(* IEC 61131-3 sources: STruCpp/tests/st-validation/data_types, 28 files *)

(* ---- string_conversions.st ---- *)
FUNCTION_BLOCK StringConversions
  VAR_OUTPUT
    (* STRING numeric parsers — strtol / strtoul / strtod under the hood,
       so `'3.14'` parses to 3 as an integer (strtol stops at the '.')
       and to 3.14 as a REAL. *)
    str_to_uint    : UINT;
    str_to_int     : INT;
    str_to_dint    : DINT;
    str_to_lint    : LINT;
    str_to_real    : REAL;
    str_to_lreal   : LREAL;
    str_negative   : INT;
    str_hex_skip   : UINT;
    str_bool_true  : BOOL;
    str_bool_false : BOOL;

    (* WSTRING numeric parsers — route through WSTRING_TO_STRING so the
       parse rules stay byte-identical with the STRING path.  Anything
       beyond the ASCII numeric subset is the user's responsibility
       (the transcoder truncates to the low byte). *)
    wstr_to_uint : UINT;
    wstr_to_real : LREAL;
    wstr_to_bool : BOOL;
  END_VAR
  VAR
    s_pi      : STRING := '3.14';
    s_half    : STRING := '4.5';
    s_neg     : STRING := '-42';
    s_trail   : STRING := '12abc';
    s_true    : STRING := 'TRUE';
    s_false   : STRING := 'no';
    ws_pi     : WSTRING := "3.14";
    ws_true   : WSTRING := "true";
  END_VAR

  str_to_uint    := TO_UINT(s_pi);     (* 3   — strtoul stops at '.' *)
  str_to_int     := TO_INT(s_pi);      (* 3 *)
  str_to_dint    := TO_DINT(s_pi);     (* 3 *)
  str_to_lint    := TO_LINT(s_pi);     (* 3 *)
  (* `3.14` round-trips bit-exact through LREAL (double) but loses
     precision narrowing to REAL (float).  Test framework's ASSERT_EQ
     does bit-exact float compare, so use an exactly-representable
     fraction here (`4.5` = 9/2 = exact in IEEE-754) instead of `3.14`. *)
  str_to_real    := TO_REAL(s_half);   (* 4.5 *)
  str_to_lreal   := TO_LREAL(s_pi);    (* 3.14 *)
  str_negative   := TO_INT(s_neg);     (* -42 *)
  str_hex_skip   := TO_UINT(s_trail);  (* 12  — strtoul stops at 'a' *)
  str_bool_true  := TO_BOOL(s_true);   (* TRUE *)
  str_bool_false := TO_BOOL(s_false);  (* FALSE *)

  wstr_to_uint := TO_UINT(ws_pi);    (* 3 *)
  wstr_to_real := TO_LREAL(ws_pi);   (* 3.14 *)
  wstr_to_bool := TO_BOOL(ws_true);  (* TRUE *)
END_FUNCTION_BLOCK

(* ---- strings.st ---- *)
FUNCTION_BLOCK StringHolder
  VAR_OUTPUT
    dblQuote : STRING;
    apostrophe : STRING;
    backslash : STRING;
    dblQuoteLen : INT;
    apostropheLen : INT;
    backslashLen : INT;
  END_VAR
  dblQuote := 'say "hello"';
  apostrophe := 'it''s working';
  backslash := 'C:\\Users\\test';
  dblQuoteLen := LEN(dblQuote);
  apostropheLen := LEN(apostrophe);
  backslashLen := LEN(backslash);
END_FUNCTION_BLOCK

(* ---- time_types.st ---- *)
FUNCTION_BLOCK TimeConversions
  VAR_OUTPUT
    (* TIME → integer scales ns→ms *)
    ms_via_dint  : DINT;
    ms_via_uint  : UINT;
    ms_via_real  : REAL;

    (* Explicit TIME_TO_<unit> helpers still work and pick the unit
       the user names, regardless of the generic TO_<int>(TIME) ms
       default.  TIME_TO_US returns LINT (int64_t) on the runtime
       side — declared wide enough to receive the raw value without
       a narrowing assignment.  Names are prefixed `unit_` so they
       don't shadow the runtime helper names on the RHS. *)
    unit_us      : LINT;
    unit_seconds : LREAL;

    (* TOD → integer scales ns→ms (since midnight) *)
    tod_ms       : DINT;

    (* DT → integer is SECONDS since 1970-01-01, matching CODESYS:
       DT_TO_DINT(DT#2019-9-1-12:0:0.0) = 1567339200.  Kept in LINT so the
       assertion reads the value rather than a truncation of it. *)
    dt_seconds   : LINT;

    (* DATE → integer is SECONDS too — CODESYS keeps DATE in DT's memory
       format, so DATE_TO_DINT(D#1970-1-2) = 86400, not 1.  UDINT rather
       than UINT: a day count fits 16 bits, a second count does not, and
       the old UINT declaration was quietly asserting a 16-bit truncation. *)
    date_seconds : UDINT;
  END_VAR
  VAR
    duration : TIME := T#1500ms;
    midpoint : TOD  := TOD#06:00:00;
    moment   : DT   := DT#1970-01-01-00:00:01;
    day      : DATE := DATE#1970-01-15;
  END_VAR

  ms_via_dint  := TIME_TO_DINT(duration);   (* 1500 *)
  ms_via_uint  := TIME_TO_UINT(duration);   (* 1500 *)
  ms_via_real  := TIME_TO_REAL(duration);   (* 1500.0 *)
  unit_us      := TIME_TO_US(duration);     (* 1_500_000 *)
  unit_seconds := TIME_TO_S(duration);      (* 1.5 *)

  tod_ms    := TOD_TO_DINT(midpoint);   (* 21_600_000 — 6h in ms *)
  dt_seconds   := TO_LINT(moment);      (* 1 — one second after the epoch *)
  date_seconds := TO_UDINT(day);        (* 1209600 — 14 days, in seconds *)
END_FUNCTION_BLOCK

(* ---- arrays.st ---- *)
TYPE IntArray : ARRAY[1..5] OF INT; END_TYPE

PROGRAM ArrayTest
  VAR
    arr : IntArray;
    sum : INT;
    first : INT;
    last : INT;
    i : INT;
  END_VAR

  (* Initialize array *)
  FOR i := 1 TO 5 DO
    arr[i] := i * 10;
  END_FOR;

  first := arr[1];
  last := arr[5];

  (* Sum all elements *)
  sum := 0;
  FOR i := 1 TO 5 DO
    sum := sum + arr[i];
  END_FOR;
END_PROGRAM

(* ---- booleans.st ---- *)
PROGRAM BooleanTypeTest
  VAR
    t : BOOL;
    f : BOOL;
    and_tt : BOOL;
    and_tf : BOOL;
    or_ff : BOOL;
    or_tf : BOOL;
    not_t : BOOL;
    not_f : BOOL;
  END_VAR

  t := TRUE;
  f := FALSE;
  and_tt := t AND t;
  and_tf := t AND f;
  or_ff := f OR f;
  or_tf := t OR f;
  not_t := NOT t;
  not_f := NOT f;
END_PROGRAM

(* ---- enum_bare_members.st ---- *)
TYPE
  TrafficState : (RED, YELLOW, GREEN);
  PedestrianState : (WALK, DONT_WALK, FLASHING);
END_TYPE

PROGRAM EnumBareTest
  VAR_INPUT
    ts : TrafficState := RED;
    ps : PedestrianState := WALK;
  END_VAR
  VAR
    result   : INT;
    isRed    : BOOL;
    isWalk   : BOOL;
  END_VAR

  (* Bare enum comparison *)
  isRed := (ts = RED);
  isWalk := (ps = WALK);

  (* CASE with bare enum labels *)
  CASE ts OF
    RED:
      result := 1;
    GREEN:
      result := 2;
    YELLOW:
      result := 3;
  END_CASE;
END_PROGRAM

(* ---- enum_dot_notation.st ---- *)
TYPE
  TrafficState : (RED, YELLOW, GREEN);
  PedestrianState : (WALK, DONT_WALK, FLASHING);
END_TYPE

PROGRAM EnumDotTest
  VAR_INPUT
    ts : TrafficState := TrafficState.RED;
    ps : PedestrianState := PedestrianState.WALK;
  END_VAR
  VAR
    result   : INT;
    isRed    : BOOL;
    isWalk   : BOOL;
  END_VAR

  (* Enum comparison with dot notation *)
  isRed := (ts = TrafficState.RED);
  isWalk := (ps = PedestrianState.WALK);

  (* CASE with enum dot-notation labels *)
  CASE ts OF
    TrafficState.RED:
      result := 1;
    TrafficState.GREEN:
      result := 2;
    TrafficState.YELLOW:
      result := 3;
  END_CASE;
END_PROGRAM

(* ---- enums.st ---- *)
TYPE
  TrafficLight : (RED, YELLOW, GREEN);
  MachineState : INT (IDLE := 0, RUNNING := 1, STOPPED := 2);
END_TYPE

PROGRAM EnumTest
  VAR
    lightDeclared : BOOL;
    stateDeclared : BOOL;
  END_VAR
  lightDeclared := TRUE;
  stateDeclared := TRUE;
END_PROGRAM

(* ---- integers.st ---- *)
PROGRAM IntegerTest
  VAR
    int_val : INT;
    dint_val : DINT;
    uint_val : UINT;
    add_result : INT;
    sub_result : INT;
  END_VAR

  int_val := 1000;
  dint_val := 100000;
  uint_val := 65000;
  add_result := 100 + 200;
  sub_result := 50 - 100;
END_PROGRAM

(* ---- multidim_arrays.st ---- *)
TYPE
  Matrix3x3 : ARRAY[0..2, 0..2] OF INT;
  OffsetArray : ARRAY[3..7] OF INT;
  OneBasedArray : ARRAY[1..5] OF INT;
  Matrix4x4 : ARRAY[1..4, 1..4] OF INT;
  Row5 : ARRAY[1..5] OF INT;
END_TYPE

PROGRAM MultidimTest
  VAR
    m : Matrix3x3;
    offArr : OffsetArray;
    oneArr : OneBasedArray;
    identity : Matrix4x4;
    row : Row5;
    i : INT;
    j : INT;
    mResult : INT;
    offResult : INT;
    oneResult : INT;
    diagSum : INT;
    mixedResult : INT;
  END_VAR

  (* 2D array access *)
  m[1, 2] := 42;
  mResult := m[1, 2];

  (* Non-zero-based array *)
  offArr[5] := 99;
  offResult := offArr[5];

  (* 1-based array *)
  FOR i := 1 TO 5 DO
    oneArr[i] := i * 10;
  END_FOR;
  oneResult := oneArr[3];

  (* Identity matrix via nested FOR *)
  FOR i := 1 TO 4 DO
    FOR j := 1 TO 4 DO
      IF i = j THEN
        identity[i, j] := 1;
      ELSE
        identity[i, j] := 0;
      END_IF;
    END_FOR;
  END_FOR;
  diagSum := identity[1, 1] + identity[2, 2] + identity[3, 3] + identity[4, 4];

  (* Mixed 1D bracket and 2D call syntax *)
  row[1] := 10;
  row[2] := 20;
  mixedResult := row[1] + row[2];
END_PROGRAM

(* ---- reals.st ---- *)
PROGRAM RealTest
  VAR
    r_add : REAL;
    r_sub : REAL;
    r_mul : REAL;
    r_div : REAL;
    r_neg : REAL;
    lr_val : LREAL;
  END_VAR

  r_add := 1.5 + 2.5;
  r_sub := 10.0 - 3.5;
  r_mul := 2.0 * 3.5;
  r_div := 10.0 / 4.0;
  r_neg := -5.5;
  lr_val := 1.23456789;
END_PROGRAM

(* ---- structs.st ---- *)
TYPE Point :
  STRUCT
    x : INT;
    y : INT;
  END_STRUCT;
END_TYPE

PROGRAM StructTest
  VAR
    p : Point;
    sum : INT;
  END_VAR

  p.x := 10;
  p.y := 20;
  sum := p.x + p.y;
END_PROGRAM

(* ---- subranges.st ---- *)
TYPE SmallInt : INT(0..100); END_TYPE

PROGRAM SubrangeTest
  VAR
    val : SmallInt;
    result : INT;
  END_VAR

  val := 50;
  result := val + 10;
END_PROGRAM

(* ---- test_arrays.st ---- *)
TEST 'Array first element'
  VAR uut : ArrayTest; END_VAR
  uut();
  ASSERT_EQ(uut.first, 10);
END_TEST

TEST 'Array last element'
  VAR uut : ArrayTest; END_VAR
  uut();
  ASSERT_EQ(uut.last, 50);
END_TEST

TEST 'Array sum of elements'
  VAR uut : ArrayTest; END_VAR
  uut();
  ASSERT_EQ(uut.sum, 150);
END_TEST

(* ---- test_booleans.st ---- *)
TEST 'TRUE AND TRUE = TRUE'
  VAR uut : BooleanTypeTest; END_VAR
  uut();
  ASSERT_TRUE(uut.and_tt);
END_TEST

TEST 'TRUE AND FALSE = FALSE'
  VAR uut : BooleanTypeTest; END_VAR
  uut();
  ASSERT_FALSE(uut.and_tf);
END_TEST

TEST 'FALSE OR FALSE = FALSE'
  VAR uut : BooleanTypeTest; END_VAR
  uut();
  ASSERT_FALSE(uut.or_ff);
END_TEST

TEST 'TRUE OR FALSE = TRUE'
  VAR uut : BooleanTypeTest; END_VAR
  uut();
  ASSERT_TRUE(uut.or_tf);
END_TEST

TEST 'NOT TRUE = FALSE'
  VAR uut : BooleanTypeTest; END_VAR
  uut();
  ASSERT_FALSE(uut.not_t);
END_TEST

TEST 'NOT FALSE = TRUE'
  VAR uut : BooleanTypeTest; END_VAR
  uut();
  ASSERT_TRUE(uut.not_f);
END_TEST

(* ---- test_enum_bare_members.st ---- *)
TEST 'Bare enum default and comparison'
  VAR uut : EnumBareTest; END_VAR
  uut();
  ASSERT_TRUE(uut.isRed, 'bare RED default should match');
  ASSERT_TRUE(uut.isWalk, 'bare WALK default should match');
END_TEST

TEST 'CASE with bare enum labels'
  VAR uut : EnumBareTest; END_VAR
  uut();
  ASSERT_EQ(uut.result, 1, 'CASE should match bare RED and set result to 1');
END_TEST

TEST 'Bare enum reassignment changes CASE branch'
  VAR uut : EnumBareTest; END_VAR

  uut.ts := GREEN;
  uut();
  ASSERT_EQ(uut.result, 2, 'GREEN -> result 2');

  uut.ts := YELLOW;
  uut();
  ASSERT_EQ(uut.result, 3, 'YELLOW -> result 3');

  uut.ts := RED;
  uut();
  ASSERT_EQ(uut.result, 1, 'RED -> result 1');
END_TEST

TEST 'Bare and qualified produce same result'
  VAR uut : EnumBareTest; END_VAR

  uut.ts := TrafficState.GREEN;
  uut();
  ASSERT_EQ(uut.result, 2, 'Qualified GREEN -> 2');

  uut.ts := GREEN;
  uut();
  ASSERT_EQ(uut.result, 2, 'Bare GREEN -> 2 (same)');
END_TEST

(* ---- test_enum_dot_notation.st ---- *)
TEST 'Enum default value and comparison with dot notation'
  VAR uut : EnumDotTest; END_VAR
  uut();
  ASSERT_TRUE(uut.isRed, 'TrafficState.RED default should match');
  ASSERT_TRUE(uut.isWalk, 'PedestrianState.WALK default should match');
END_TEST

TEST 'CASE with enum dot-notation labels'
  VAR uut : EnumDotTest; END_VAR
  uut();
  ASSERT_EQ(uut.result, 1, 'CASE should match TrafficState.RED and set result to 1');
END_TEST

TEST 'Enum reassignment changes CASE branch'
  VAR uut : EnumDotTest; END_VAR

  uut.ts := TrafficState.GREEN;
  uut();
  ASSERT_EQ(uut.result, 2, 'GREEN -> result 2');

  uut.ts := TrafficState.YELLOW;
  uut();
  ASSERT_EQ(uut.result, 3, 'YELLOW -> result 3');

  uut.ts := TrafficState.RED;
  uut();
  ASSERT_EQ(uut.result, 1, 'RED -> result 1');
END_TEST

(* ---- test_enums.st ---- *)
TEST 'Enum type declarations compile and program runs'
  VAR uut : EnumTest; END_VAR
  uut();
  ASSERT_TRUE(uut.lightDeclared);
  ASSERT_TRUE(uut.stateDeclared);
END_TEST

(* ---- test_integers.st ---- *)
TEST 'INT holds 1000'
  VAR uut : IntegerTest; END_VAR
  uut();
  ASSERT_EQ(uut.int_val, 1000);
END_TEST

TEST 'DINT holds 100000'
  VAR uut : IntegerTest; END_VAR
  uut();
  ASSERT_EQ(uut.dint_val, 100000);
END_TEST

TEST 'UINT holds 65000'
  VAR uut : IntegerTest; END_VAR
  uut();
  ASSERT_EQ(uut.uint_val, 65000);
END_TEST

TEST 'Integer addition'
  VAR uut : IntegerTest; END_VAR
  uut();
  ASSERT_EQ(uut.add_result, 300);
END_TEST

TEST 'Integer subtraction produces negative'
  VAR uut : IntegerTest; END_VAR
  uut();
  ASSERT_EQ(uut.sub_result, -50);
END_TEST

(* ---- test_multidim_arrays.st ---- *)
TEST '2D array access'
  VAR uut : MultidimTest; END_VAR
  uut();
  ASSERT_EQ(uut.mResult, 42);
END_TEST

TEST 'Non-zero-based array ARRAY[3..7]'
  VAR uut : MultidimTest; END_VAR
  uut();
  ASSERT_EQ(uut.offResult, 99);
END_TEST

TEST '1-based array ARRAY[1..5]'
  VAR uut : MultidimTest; END_VAR
  uut();
  ASSERT_EQ(uut.oneResult, 30);
END_TEST

TEST 'Identity matrix via nested FOR loops'
  VAR uut : MultidimTest; END_VAR
  uut();
  ASSERT_EQ(uut.diagSum, 4);
END_TEST

TEST 'Mixed 1D and 2D access'
  VAR uut : MultidimTest; END_VAR
  uut();
  ASSERT_EQ(uut.mixedResult, 30);
END_TEST

(* ---- test_reals.st ---- *)
TEST 'REAL addition'
  VAR uut : RealTest; END_VAR
  uut();
  ASSERT_NEAR(uut.r_add, 4.0, 0.001);
END_TEST

TEST 'REAL subtraction'
  VAR uut : RealTest; END_VAR
  uut();
  ASSERT_NEAR(uut.r_sub, 6.5, 0.001);
END_TEST

TEST 'REAL multiplication'
  VAR uut : RealTest; END_VAR
  uut();
  ASSERT_NEAR(uut.r_mul, 7.0, 0.001);
END_TEST

TEST 'REAL division'
  VAR uut : RealTest; END_VAR
  uut();
  ASSERT_NEAR(uut.r_div, 2.5, 0.001);
END_TEST

TEST 'REAL negation'
  VAR uut : RealTest; END_VAR
  uut();
  ASSERT_NEAR(uut.r_neg, -5.5, 0.001);
END_TEST

TEST 'LREAL precision'
  VAR uut : RealTest; END_VAR
  uut();
  ASSERT_NEAR(uut.lr_val, 1.23456789, 0.0001);
END_TEST

(* ---- test_string_conversions.st ---- *)
(* End-to-end coverage for STRING / WSTRING → numeric conversions.
   STRING parsers route through `strtol` / `strtoul` / `strtod`; WSTRING
   parsers route through `WSTRING_TO_STRING` first so the wide path
   stays byte-identical with the narrow one.  Pin both surfaces so a
   future reroute (e.g. someone switching to a UTF-16-aware parser)
   doesn't silently change observable behaviour. *)

TEST 'TO_UINT of "3.14" stops at the dot (parses to 3)'
  VAR uut : StringConversions; END_VAR
  uut();
  ASSERT_EQ(uut.str_to_uint, 3);
END_TEST

TEST 'TO_INT of "3.14" stops at the dot (parses to 3)'
  VAR uut : StringConversions; END_VAR
  uut();
  ASSERT_EQ(uut.str_to_int, 3);
END_TEST

TEST 'TO_DINT of "3.14" stops at the dot (parses to 3)'
  VAR uut : StringConversions; END_VAR
  uut();
  ASSERT_EQ(uut.str_to_dint, 3);
END_TEST

TEST 'TO_LINT of "3.14" stops at the dot (parses to 3)'
  VAR uut : StringConversions; END_VAR
  uut();
  ASSERT_EQ(uut.str_to_lint, 3);
END_TEST

TEST 'TO_REAL of "4.5" parses the fraction (bit-exact via REAL)'
  VAR uut : StringConversions; END_VAR
  uut();
  ASSERT_EQ(uut.str_to_real, 4.5);
END_TEST

TEST 'TO_LREAL of "3.14" parses the fraction at LREAL precision'
  VAR uut : StringConversions; END_VAR
  uut();
  ASSERT_EQ(uut.str_to_lreal, 3.14);
END_TEST

TEST 'TO_INT of "-42" parses the sign'
  VAR uut : StringConversions; END_VAR
  uut();
  ASSERT_EQ(uut.str_negative, -42);
END_TEST

TEST 'TO_UINT of "12abc" stops at the first non-digit (parses to 12)'
  VAR uut : StringConversions; END_VAR
  uut();
  ASSERT_EQ(uut.str_hex_skip, 12);
END_TEST

TEST 'TO_BOOL of "TRUE" returns TRUE'
  VAR uut : StringConversions; END_VAR
  uut();
  ASSERT_EQ(uut.str_bool_true, TRUE);
END_TEST

TEST 'TO_BOOL of "no" returns FALSE'
  VAR uut : StringConversions; END_VAR
  uut();
  ASSERT_EQ(uut.str_bool_false, FALSE);
END_TEST

TEST 'WSTRING TO_UINT of "3.14" parses to 3 (matches STRING surface)'
  VAR uut : StringConversions; END_VAR
  uut();
  ASSERT_EQ(uut.wstr_to_uint, 3);
END_TEST

TEST 'WSTRING TO_LREAL of "3.14" parses to 3.14 (matches STRING surface)'
  VAR uut : StringConversions; END_VAR
  uut();
  ASSERT_EQ(uut.wstr_to_real, 3.14);
END_TEST

TEST 'WSTRING TO_BOOL of "true" returns TRUE'
  VAR uut : StringConversions; END_VAR
  uut();
  ASSERT_EQ(uut.wstr_to_bool, TRUE);
END_TEST

(* ---- test_strings.st ---- *)
TEST 'Double-quotes inside string preserved'
  VAR sh : StringHolder; END_VAR
  sh();
  ASSERT_EQ(sh.dblQuoteLen, 11);
END_TEST

TEST 'Doubled single-quotes become apostrophe'
  VAR sh : StringHolder; END_VAR
  sh();
  ASSERT_EQ(sh.apostropheLen, 12);
END_TEST

TEST 'Backslashes preserved in string'
  VAR sh : StringHolder; END_VAR
  sh();
  ASSERT_EQ(sh.backslashLen, 15);
END_TEST

(* ---- test_structs.st ---- *)
TEST 'Struct member access'
  VAR uut : StructTest; END_VAR
  uut();
  ASSERT_EQ(uut.p.x, 10);
  ASSERT_EQ(uut.p.y, 20);
END_TEST

TEST 'Struct member arithmetic'
  VAR uut : StructTest; END_VAR
  uut();
  ASSERT_EQ(uut.sum, 30);
END_TEST

(* ---- test_subranges.st ---- *)
TEST 'Subrange assignment and arithmetic'
  VAR uut : SubrangeTest; END_VAR
  uut();
  ASSERT_EQ(uut.result, 60);
END_TEST

(* ---- test_time_types.st ---- *)
(* Regression suite for the temporal-to-numeric scaling fix.
   The original bug: TO_UINT(T#5s) returned the low 16 bits of the
   nanosecond count (61952) instead of the expected ms count (5000).
   Codegen wraps temporal args with a unit helper before the integer
   cast.  The unit is CODESYS's, per type: milliseconds for TIME and
   TOD, seconds for DT and DATE (DOPE-618).  These tests pin every
   elementary temporal source so the scaling can't silently regress. *)

TEST 'TIME_TO_DINT returns milliseconds'
  VAR uut : TimeConversions; END_VAR
  uut();
  ASSERT_EQ(uut.ms_via_dint, 1500);
END_TEST

TEST 'TIME_TO_UINT returns milliseconds (low 16 bits when overflowing)'
  VAR uut : TimeConversions; END_VAR
  uut();
  ASSERT_EQ(uut.ms_via_uint, 1500);
END_TEST

TEST 'TIME_TO_REAL returns milliseconds as float'
  VAR uut : TimeConversions; END_VAR
  uut();
  ASSERT_EQ(uut.ms_via_real, 1500.0);
END_TEST

TEST 'TIME_TO_US returns microseconds (explicit helper, not codegen wrap)'
  VAR uut : TimeConversions; END_VAR
  uut();
  ASSERT_EQ(uut.unit_us, 1500000);
END_TEST

TEST 'TIME_TO_S returns seconds as float'
  VAR uut : TimeConversions; END_VAR
  uut();
  ASSERT_EQ(uut.unit_seconds, 1.5);
END_TEST

TEST 'TOD_TO_DINT returns milliseconds since midnight'
  VAR uut : TimeConversions; END_VAR
  uut();
  ASSERT_EQ(uut.tod_ms, 21600000);
END_TEST

TEST 'DT_TO_LINT returns seconds since epoch, as CODESYS does'
  VAR uut : TimeConversions; END_VAR
  uut();
  (* Was 1000 (milliseconds) before DOPE-618.  CODESYS holds DT in seconds:
     DT_TO_DINT(DT#2019-9-1-12:0:0.0) = 1567339200. *)
  ASSERT_EQ(uut.dt_seconds, 1);
END_TEST

TEST 'DATE_TO_UDINT returns seconds since 1970-01-01, as CODESYS does'
  VAR uut : TimeConversions; END_VAR
  uut();
  (* Was 14 (a day count) before DOPE-618.  CODESYS keeps DATE in DT's
     memory format: DATE_TO_DINT(D#1970-1-2) = 86400, not 1.  This is why
     every OSCAT DATE helper divided by 86400 and got zero. *)
  ASSERT_EQ(uut.date_seconds, 1209600);
END_TEST

(* ---- test_type_aliases.st ---- *)
TEST 'MyInt alias works like INT'
  VAR uut : TypeAliasTest; END_VAR
  uut();
  ASSERT_EQ(uut.intResult, 50);
END_TEST

TEST 'MyReal alias works like REAL'
  VAR uut : TypeAliasTest; END_VAR
  uut();
  ASSERT_NEAR(uut.realResult, 6.28, 0.01);
END_TEST

(* ---- type_aliases.st ---- *)
TYPE
  MyInt : INT;
  MyReal : REAL;
END_TYPE

PROGRAM TypeAliasTest
  VAR
    a : MyInt;
    b : MyReal;
    intResult : INT;
    realResult : REAL;
  END_VAR
  a := 42;
  b := 3.14;
  intResult := a + 8;
  realResult := b * 2.0;
END_PROGRAM
